{attribute 'qualified_only'}
VAR_GLOBAL
	_DI				AT %I*: 	U_IN_IO_Translate;
	ANALOG			AT %I*:		ARRAY[1..4] OF INT;	// Temperature module
	
END_VAR

(* stored: Version 1.1.0.1, ProductVersion 3.1.4024.10
   GVL IN: Id {c44d48c9-f66f-4539-acb1-5e7a1a17ef6b} *)
